(* CODESYS project 3.1GearTest.project

Project tree, tasks and I/O mapping:
  Device : CODESYS SoftMotion Win V3 x64, 3S - Smart Software Solutions GmbH, version 3.5.12.0
    application Application
      libraries: Standard, * (System); VisuDialogs, * (System)
      task MainTask (cyclic, interval t#2ms, priority 1) calls PLC_PRG
      task VISU_TASK (cyclic, interval 100 ms, priority 31) calls VisuElems.Visu_Prg
      program PLC_PRG [ST]
      visualisation Visualization
      trace Trace (task MainTask): AxisMaster.fActVelocity, AxisSlave.fActVelocity, AxisMaster.fActPosition, AxisSlave.fActPosition, AxisMaster.fActAcceleration, AxisSlave.fActAcceleration, PLC_PRG.mcGearInPos.Execute, PLC_PRG.mcGearInPos.InSync, PLC_PRG.mcGearInPos.Busy, PLC_PRG.mcGearInPos.StartSync, AxisMaster.fSetPosition, AxisSlave.fSetPosition
    SoftMotion General Axis Pool
      AxisMaster : SM_Drive_Virtual, 3S - Smart Software Solutions GmbH, order no. 1805, version 4.0.0.0
          settings: wDriveID = 0; iMovementType = 0
      AxisSlave : SM_Drive_Virtual, 3S - Smart Software Solutions GmbH, order no. 1805, version 4.0.0.0
          settings: iMovementType = 0
  text list GlobalTextList
  text list AxisStatus
*)

// Device/Application/PLC_PRG
PROGRAM PLC_PRG
VAR
	//定义Master主轴相关的功能块
	mcPMaster  		:  MC_Power ;
	mcMoveVelocity  : MC_MoveVelocity ;
	mcStopMaster  	: MC_stop;
	mcResetM         : MC_Reset;
	//定义从轴相关功能块；
	mcPSlave    : MC_Power ;
	mcStopSlave : MC_Stop ;
	mcResetS      : MC_Reset;
	mcSetPostion  : MC_SetPosition;
	//Gear 
	mcGearIn  	: MC_GearIn ;
	mcGearOut  	: MC_GearOut ;
	mcGearInPos : MC_GearInPos;
	//辅助变量
	bGearIn   	: BOOL;
	bStartMove  : BOOL;
END_VAR

//主轴和从轴的使能
mcPMaster(
	Axis:= AxisMaster, 
	Enable:= TRUE , 
	bRegulatorOn:= TRUE , 
	bDriveStart:=TRUE , 
	Status=> , 
	bRegulatorRealState=> , 
	bDriveStartRealState=> , 
	Busy=> , 
	Error=> , 
	ErrorID=> );
mcPSlave(
	Axis:= AxisSlave , 
	Enable:= TRUE, 
	bRegulatorOn:= TRUE , 
	bDriveStart:= TRUE, 
	Status=> , 
	bRegulatorRealState=> , 
	bDriveStartRealState=> , 
	Busy=> , 
	Error=> , 
	ErrorID=> );
//齿轮耦合
mcGearIn(
	Master:= AxisMaster, 
	Slave:= AxisSlave, 
	Execute:= , 
	RatioNumerator:= , 
	RatioDenominator:= , 
	Acceleration:= , 
	Deceleration:= , 
	Jerk:= , 
	InGear=> , 
	Busy=> , 
	CommandAborted=> , 
	Error=> , 
	ErrorID=> );
mcGearInPos(
	Master:= AxisMaster, 
	Slave:= AxisSlave, 
	Execute:= , 
	RatioNumerator:= , 
	RatioDenominator:= , 
	MasterSyncPosition:= , 
	SlaveSyncPosition:= , 
	MasterStartDistance:= , 
	AvoidReversal:= , 
	StartSync=> , 
	InSync=> , 
	Busy=> , 
	CommandAborted=> , 
	Error=> , 
	ErrorID=> );
mcGearOut(
	Slave:=AxisSlave , 
	Execute:= , 
	Done=> , 
	Busy=> , 
	Error=> , 
	ErrorID=> );	
//主轴开始运动
mcMoveVelocity(
	Axis:=AxisMaster , 
	Execute:=  , 
	Velocity:= , 
	Acceleration:= 100, 
	Deceleration:= 100, 
	Jerk:= , 
	Direction:= , 
	InVelocity=> , 
	Busy=> , 
	CommandAborted=> , 
	Error=> , 
	ErrorID=> );
	
//停止
mcStopMaster(
	Axis:= AxisMaster, 
	Execute:= , 
	Deceleration:= , 
	Jerk:= , 
	Done=> , 
	Busy=> , 
	Error=> , 
	ErrorID=> );
mcStopSlave(
	Axis:= AxisSlave, 
	Execute:= , 
	Deceleration:= , 
	Jerk:= , 
	Done=> , 
	Busy=> , 
	Error=> , 
	ErrorID=> );
mcSetPostion(
	Axis:= AxisSlave, 
	Execute:= , 
	Position:= , 
	Mode:= , 
	Done=> , 
	Busy=> , 
	Error=> , 
	ErrorID=> );	
//复位
mcResetM(
	Axis:= AxisMaster, 
	Execute:= , 
	Done=> , 
	Busy=> , 
	Error=> , 
	ErrorID=> );
mcResetS(
	Axis:= AxisSlave, 
	Execute:= , 
	Done=> , 
	Busy=> , 
	Error=> , 
	ErrorID=> );

END_PROGRAM

// Device/Application/Visualization
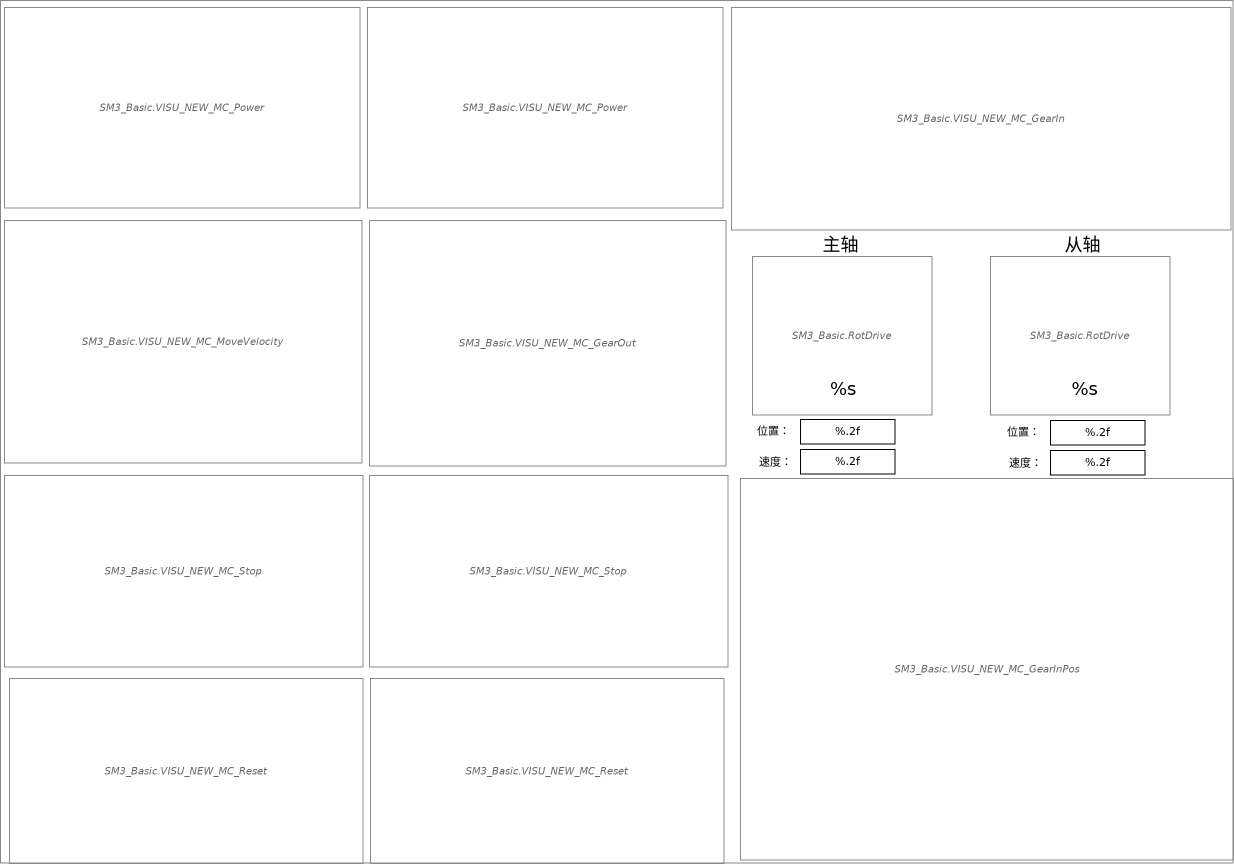
VISUALIZATION Visualization  // 1234x864
    Frame (4,7 356x201)
        shows SM3_Basic.VISU_NEW_MC_Power(m_Input_FB := PLC_PRG.mcPMaster)
    Frame (367,7 356x201)
        shows SM3_Basic.VISU_NEW_MC_Power(m_Input_FB := PLC_PRG.mcPSlave)
    Frame (4,220 358x243)
        shows SM3_Basic.VISU_NEW_MC_MoveVelocity(m_Input_FB := PLC_PRG.mcMoveVelocity)
    Frame (4,475 359x192)
        shows SM3_Basic.VISU_NEW_MC_Stop(m_Input_FB := PLC_PRG.mcStopMaster)
    Frame (369,475 359x192)
        shows SM3_Basic.VISU_NEW_MC_Stop(m_Input_FB := PLC_PRG.mcStopSlave)
    Frame (369,220 357x246)
        shows SM3_Basic.VISU_NEW_MC_GearOut(m_Input_FB := PLC_PRG.mcGearOut)
    Frame (731,7 500x223)
        shows SM3_Basic.VISU_NEW_MC_GearIn(m_Input_FB := PLC_PRG.mcGearIn)
    Frame (752,256 180x159)
        shows SM3_Basic.RotDrive(m_Input_AXISREF := Axismaster)
    Frame (990,256 180x159)
        shows SM3_Basic.RotDrive(m_Input_AXISREF := AxisSlave)
    Frame (9,678 354x186)
        shows SM3_Basic.VISU_NEW_MC_Reset(m_Input_FB := PLC_PRG.mcResetM)
    Frame (370,678 354x186)
        shows SM3_Basic.VISU_NEW_MC_Reset(m_Input_FB := PLC_PRG.mcResetS)
    Frame (740,478 494x382)
        shows SM3_Basic.VISU_NEW_MC_GearInPos(m_Input_FB := PLC_PRG.mcGearInPos)
    Label (793,230 95x30), "主轴"
    Label (1035,230 95x30), "从轴"
    Label (734,416 79x30), "位置："
    Label (736,447 79x30), "速度："
    Rectangle (800,419 95x25), "%.2f", text variable: AxisMaster.fActPosition
    Rectangle (800,449 95x25), "%.2f", text variable: AxisMaster.fActVelocity
    Label (986,448 79x30), "速度："
    Label (984,417 79x30), "位置："
    Rectangle (1050,420 95x25), "%.2f", text variable: AxisSlave.fActPosition
    Rectangle (1050,450 95x25), "%.2f", text variable: AxisSlave.fActVelocity
    Rectangle (738,374 211x30), "%s", text list: 'AxisStatus', text index: AxisMaster.nAxisState
    Rectangle (978,374 214x30), "%s", text list: 'AxisStatus', text index: AxisSlave.nAxisState
END_VISUALIZATION

(* text list AxisStatus (id | default)
  0 | power_off
  1 | errorstop
  2 | stopping
  3 | standstill
  4 | discrete_motion
  5 | continuous_motion
  6 | synchronized_motion
  7 | homing
   |  *)
